INTERFACE I_HostContent EXTENDS __SYSTEM.IQueryInterface

METHOD AddContent
VAR_INPUT
	Content : I_Content;
END_VAR
END_METHOD

METHOD AddDataAsContent : I_Content;
VAR_INPUT
	Name : T_MAXSTRING;
	Data : I_Datatype;
END_VAR
END_METHOD

METHOD PUBLIC TryGetContentByName : BOOL
VAR_INPUT
	Name : T_MAXSTRING;
	Destination : REFERENCE TO I_Content;
END_VAR
END_METHOD

END_INTERFACE

(* stored: Version 1.1.0.1, ProductVersion 3.1.4024.12
   Itf I_HostContent: Id {b6826600-a2aa-01de-2bb0-f4ea403d72a8}
   Method AddContent: Id {cf987282-ff3f-0893-1bfe-87351ab41c96}
   Method AddDataAsContent: Id {794f70b3-ebc0-4576-8112-4da844755c3b}
   Method TryGetContentByName: Id {c3b2381b-d905-05c0-2520-a309855441a7} *)
